TYPE DUT_SENSOR_DATAS_h5 :
UNION
	data_lreal:REAL;
	data_byte:ARRAY[0..3] OF BYTE;
END_UNION
END_TYPE

(* stored: Version 1.1.0.1, ProductVersion 3.1.4024.6
   DUT DUT_SENSOR_DATAS_h5: Id {5d64e7ba-5924-4d16-839a-d9a8e630f0bb} *)
